{attribute 'GeneratedUsingTerminal: EL3632-0000-0016'}
{attribute addProperty BoxType "EL3632-0000-0016"}
{attribute addProperty Id "Ch1_Sample_CountAT %I*UINT2"}
{attribute addProperty CRC "3260899128"}
{attribute addProperty Size "2"}
TYPE Sample_Count_C25D5F38 :
STRUCT
	{attribute addProperty Name "Ch1_Sample_Count"}
	Ch1_Sample_Count AT %I* : UINT;
END_STRUCT
END_TYPE

(* stored: Version 1.2.0.0, ProductVersion 3.1.4024.9
   DUT Sample_Count_C25D5F38: Id {2791db7b-a913-4028-b7b5-b42e3e756c29} *)
